FUNCTION Buffer_Layout_Set_DInt_Array : UINT
VAR_INPUT
END_VAR
VAR
END_VAR

END_FUNCTION

(* stored: Version 1.1.0.1, ProductVersion 3.1.4024.10
   POU Buffer_Layout_Set_DInt_Array: Id {c84beb60-a381-45ad-90ab-ad5ab2827468}, SpecialFunc None *)
